Staubli VAL3: loopMode.pgx

public program loopMode()
  local num i
  local string sSwapLoad
  local num nSwapTotal
  local num l_nSize
begin
  //  set the process list after one cycle done
  //
  //  the variable loadProg has to not be minus than 1 items
  //  THIS IS THE NO LOOP CODE
  //
  if !saveCycle:bLoop
    //
    call delete(0,1)
  else
    //
    //  LOOP MODE
    //
    call getSize(l_nSize,1)
    if cycleStatus:nProg<l_nSize-1
      // continue
      cycleStatus:nProg=cycleStatus:nProg+1
    else
      // REINIT
      for i=0 to l_nSize-1
        saveCycle:nDoneCycle[i]=0
      endFor
      cycleStatus:nProg=0
    endIf
  endIf
end
